(* IEC 61131-3 sources: Berechnungsplattform/PLC_CODESYS/Joystick, 2 files *)

(* ---- Gessmann_Joystick.st ---- *)
(* ============================================================================
   Gessmann Joystick / Thrust Lever CAN Interface
   Development Environment: CODESYS
   PLC Hardware: Intercontrol DIGSY Fusion S
   Description: Function block for reading Gessmann joystick and thrust lever
                signals via CAN bus
   ============================================================================ *)

TYPE Joystick_Axis :
STRUCT
    nRawValue       : INT;          (* Raw value from CAN message *)
    rScaledValue    : REAL;         (* Scaled value (-100.0 to +100.0 %) *)
    rDeadzone       : REAL := 5.0;  (* Deadzone in percent *)
    bInDeadzone     : BOOL;         (* Axis is in deadzone *)
    nMin            : INT := -32768;(* Minimum raw value *)
    nMax            : INT := 32767; (* Maximum raw value *)
    nCenter         : INT := 0;     (* Center/neutral raw value *)
END_STRUCT
END_TYPE

TYPE Gessmann_Joystick_Data :
STRUCT
    (* Axis data *)
    stAxisX         : Joystick_Axis;    (* X-Axis (left/right) *)
    stAxisY         : Joystick_Axis;    (* Y-Axis (forward/backward) *)
    stAxisZ         : Joystick_Axis;    (* Z-Axis / Twist (rotation) *)
    stThrustLever   : Joystick_Axis;    (* Thrust lever position *)

    (* Button states *)
    bButton1        : BOOL := FALSE;    (* Button 1 state *)
    bButton2        : BOOL := FALSE;    (* Button 2 state *)
    bButton3        : BOOL := FALSE;    (* Button 3 state *)
    bButton4        : BOOL := FALSE;    (* Button 4 state *)
    bButton5        : BOOL := FALSE;    (* Button 5 state *)
    bButton6        : BOOL := FALSE;    (* Button 6 state *)
    bButton7        : BOOL := FALSE;    (* Button 7 state *)
    bButton8        : BOOL := FALSE;    (* Button 8 state *)

    (* Status *)
    bOnline         : BOOL := FALSE;    (* Joystick communication active *)
    bError          : BOOL := FALSE;    (* Error flag *)
    dwErrorCode     : DWORD := 0;       (* Error code *)
END_STRUCT
END_TYPE

(* ============================================================================
   FUNCTION_BLOCK: FB_Gessmann_Joystick
   Description: Gessmann joystick/thrust lever handler via CAN
   ============================================================================ *)
FUNCTION_BLOCK FB_Gessmann_Joystick
VAR_INPUT
    bEnable             : BOOL := FALSE;        (* Enable joystick processing *)
    stCANMessage        : CAN_Message;          (* Incoming CAN message *)
    bNewCANMessage      : BOOL := FALSE;        (* New CAN message received *)
    dwJoystickCANID     : DWORD := 16#180;      (* Base CAN ID for joystick *)
    dwThrustLeverCANID  : DWORD := 16#181;      (* CAN ID for thrust lever *)
    dwButtonsCANID      : DWORD := 16#182;      (* CAN ID for buttons *)
    tTimeout            : TIME := T#500MS;      (* Communication timeout *)
    rDeadzoneX          : REAL := 5.0;          (* Deadzone for X-axis in % *)
    rDeadzoneY          : REAL := 5.0;          (* Deadzone for Y-axis in % *)
    rDeadzoneZ          : REAL := 5.0;          (* Deadzone for Z-axis in % *)
    rDeadzoneThrustLever: REAL := 2.0;          (* Deadzone for thrust lever in % *)
END_VAR

VAR_OUTPUT
    stJoystickData      : Gessmann_Joystick_Data;   (* Complete joystick data *)
    rAxisX              : REAL := 0.0;              (* X-Axis scaled output *)
    rAxisY              : REAL := 0.0;              (* Y-Axis scaled output *)
    rAxisZ              : REAL := 0.0;              (* Z-Axis scaled output *)
    rThrustLever        : REAL := 0.0;              (* Thrust lever scaled output *)
    bOnline             : BOOL := FALSE;            (* Communication status *)
    bError              : BOOL := FALSE;            (* Error flag *)
END_VAR

VAR
    tCommTimeout        : TON;                      (* Communication timeout timer *)
    bMessageReceived    : BOOL := FALSE;            (* Flag for received message *)
    dwLastMessageTime   : DWORD := 0;               (* Timestamp of last message *)
END_VAR

(* Main execution *)
IF NOT bEnable THEN
    (* Reset all outputs when disabled *)
    stJoystickData.bOnline := FALSE;
    bOnline := FALSE;
    rAxisX := 0.0;
    rAxisY := 0.0;
    rAxisZ := 0.0;
    rThrustLever := 0.0;
    RETURN;
END_IF

(* Set deadzone values *)
stJoystickData.stAxisX.rDeadzone := rDeadzoneX;
stJoystickData.stAxisY.rDeadzone := rDeadzoneY;
stJoystickData.stAxisZ.rDeadzone := rDeadzoneZ;
stJoystickData.stThrustLever.rDeadzone := rDeadzoneThrustLever;

(* Process incoming CAN messages *)
IF bNewCANMessage THEN
    bMessageReceived := TRUE;

    (* Process Joystick axes message *)
    IF stCANMessage.ID = dwJoystickCANID THEN
        (* Parse X-Axis from bytes 0-1 (high byte first)
           Using WORD intermediate to handle unsigned byte values correctly
           before converting to signed INT for the axis value *)
        stJoystickData.stAxisX.nRawValue := WORD_TO_INT(
            SHL(BYTE_TO_WORD(stCANMessage.Data[0]), 8)
            + BYTE_TO_WORD(stCANMessage.Data[1]));

        (* Parse Y-Axis from bytes 2-3 *)
        stJoystickData.stAxisY.nRawValue := WORD_TO_INT(
            SHL(BYTE_TO_WORD(stCANMessage.Data[2]), 8)
            + BYTE_TO_WORD(stCANMessage.Data[3]));

        (* Parse Z-Axis from bytes 4-5 *)
        stJoystickData.stAxisZ.nRawValue := WORD_TO_INT(
            SHL(BYTE_TO_WORD(stCANMessage.Data[4]), 8)
            + BYTE_TO_WORD(stCANMessage.Data[5]));

        (* Scale and apply deadzone to each axis *)
        ScaleAxis(stAxis := stJoystickData.stAxisX);
        ScaleAxis(stAxis := stJoystickData.stAxisY);
        ScaleAxis(stAxis := stJoystickData.stAxisZ);

        (* Update outputs *)
        rAxisX := stJoystickData.stAxisX.rScaledValue;
        rAxisY := stJoystickData.stAxisY.rScaledValue;
        rAxisZ := stJoystickData.stAxisZ.rScaledValue;

    (* Process Thrust Lever message *)
    ELSIF stCANMessage.ID = dwThrustLeverCANID THEN
        (* Parse Thrust Lever from bytes 0-1 *)
        stJoystickData.stThrustLever.nRawValue := WORD_TO_INT(
            SHL(BYTE_TO_WORD(stCANMessage.Data[0]), 8)
            + BYTE_TO_WORD(stCANMessage.Data[1]));

        (* Scale and apply deadzone *)
        ScaleAxis(stAxis := stJoystickData.stThrustLever);
        rThrustLever := stJoystickData.stThrustLever.rScaledValue;

    (* Process Buttons message *)
    ELSIF stCANMessage.ID = dwButtonsCANID THEN
        (* Parse button states from byte 0 *)
        stJoystickData.bButton1 := (stCANMessage.Data[0] AND 16#01) <> 0;
        stJoystickData.bButton2 := (stCANMessage.Data[0] AND 16#02) <> 0;
        stJoystickData.bButton3 := (stCANMessage.Data[0] AND 16#04) <> 0;
        stJoystickData.bButton4 := (stCANMessage.Data[0] AND 16#08) <> 0;
        stJoystickData.bButton5 := (stCANMessage.Data[0] AND 16#10) <> 0;
        stJoystickData.bButton6 := (stCANMessage.Data[0] AND 16#20) <> 0;
        stJoystickData.bButton7 := (stCANMessage.Data[0] AND 16#40) <> 0;
        stJoystickData.bButton8 := (stCANMessage.Data[0] AND 16#80) <> 0;
    END_IF

    (* Reset timeout timer on any valid message *)
    tCommTimeout(IN := FALSE);
END_IF

(* Communication timeout handling *)
tCommTimeout(IN := bEnable, PT := tTimeout);
IF tCommTimeout.Q THEN
    (* Timeout occurred - no message received within timeout period *)
    stJoystickData.bOnline := FALSE;
    stJoystickData.bError := TRUE;
    stJoystickData.dwErrorCode := 1; (* Timeout error *)
    bOnline := FALSE;
    bError := TRUE;

    (* Reset outputs to safe values *)
    rAxisX := 0.0;
    rAxisY := 0.0;
    rAxisZ := 0.0;
    rThrustLever := 0.0;
ELSE
    IF bMessageReceived THEN
        stJoystickData.bOnline := TRUE;
        stJoystickData.bError := FALSE;
        stJoystickData.dwErrorCode := 0;
        bOnline := TRUE;
        bError := FALSE;
    END_IF
END_IF

END_FUNCTION_BLOCK

(* ============================================================================
   ACTION: ScaleAxis
   Description: Scales raw joystick axis value to percentage and applies deadzone
   ============================================================================ *)
ACTION ScaleAxis
VAR_IN_OUT
    stAxis  : Joystick_Axis;
END_VAR

VAR
    rRawPercent : REAL;
    rRange      : REAL;
END_VAR

(* Calculate percentage from raw value *)
IF stAxis.nRawValue >= stAxis.nCenter THEN
    (* Positive direction *)
    rRange := INT_TO_REAL(stAxis.nMax - stAxis.nCenter);
    IF rRange > 0.0 THEN
        rRawPercent := INT_TO_REAL(stAxis.nRawValue - stAxis.nCenter) / rRange * 100.0;
    ELSE
        rRawPercent := 0.0;
    END_IF
ELSE
    (* Negative direction *)
    rRange := INT_TO_REAL(stAxis.nCenter - stAxis.nMin);
    IF rRange > 0.0 THEN
        rRawPercent := INT_TO_REAL(stAxis.nRawValue - stAxis.nCenter) / rRange * 100.0;
    ELSE
        rRawPercent := 0.0;
    END_IF
END_IF

(* Limit to valid range *)
IF rRawPercent > 100.0 THEN
    rRawPercent := 100.0;
ELSIF rRawPercent < -100.0 THEN
    rRawPercent := -100.0;
END_IF

(* Apply deadzone *)
IF ABS(rRawPercent) < stAxis.rDeadzone THEN
    stAxis.rScaledValue := 0.0;
    stAxis.bInDeadzone := TRUE;
ELSE
    (* Scale remaining range to full output range *)
    IF rRawPercent > 0.0 THEN
        stAxis.rScaledValue := (rRawPercent - stAxis.rDeadzone) / (100.0 - stAxis.rDeadzone) * 100.0;
    ELSE
        stAxis.rScaledValue := (rRawPercent + stAxis.rDeadzone) / (100.0 - stAxis.rDeadzone) * 100.0;
    END_IF
    stAxis.bInDeadzone := FALSE;
END_IF

END_ACTION

(* ---- Thrust_Lever_Control.st ---- *)
(* ============================================================================
   Thrust Lever Control Function Block
   Development Environment: CODESYS
   PLC Hardware: Intercontrol DIGSY Fusion S
   Description: Advanced thrust lever control with ramping, limits, and modes
   ============================================================================ *)

TYPE Thrust_Mode :
(
    THRUST_MODE_MANUAL := 0,        (* Direct joystick control *)
    THRUST_MODE_CRUISE := 1,        (* Cruise control / hold speed *)
    THRUST_MODE_RAMP := 2,          (* Ramped acceleration/deceleration *)
    THRUST_MODE_EMERGENCY := 3      (* Emergency stop *)
);
END_TYPE

TYPE Thrust_Status :
STRUCT
    eMode           : Thrust_Mode;      (* Current operating mode *)
    rCurrentThrust  : REAL;             (* Current thrust output (%) *)
    rTargetThrust   : REAL;             (* Target thrust (%) *)
    rRampRate       : REAL;             (* Current ramp rate (%/s) *)
    bLimitActive    : BOOL;             (* Limit is active *)
    bRamping        : BOOL;             (* Currently ramping *)
    bEmergency      : BOOL;             (* Emergency mode active *)
END_STRUCT
END_TYPE

(* ============================================================================
   FUNCTION_BLOCK: FB_Thrust_Lever_Control
   Description: Advanced thrust lever control with multiple operating modes
   ============================================================================ *)
FUNCTION_BLOCK FB_Thrust_Lever_Control
VAR_INPUT
    bEnable             : BOOL := FALSE;        (* Enable control *)
    rThrustLeverInput   : REAL := 0.0;          (* Raw thrust lever input (-100 to +100 %) *)
    eRequestedMode      : Thrust_Mode := THRUST_MODE_MANUAL;  (* Requested mode *)
    bEmergencyStop      : BOOL := FALSE;        (* Emergency stop trigger *)
    bCruiseSet          : BOOL := FALSE;        (* Set cruise control *)
    bCruiseResume       : BOOL := FALSE;        (* Resume cruise control *)
    bCruiseCancel       : BOOL := FALSE;        (* Cancel cruise control *)

    (* Configuration parameters *)
    rMaxThrust          : REAL := 100.0;        (* Maximum thrust limit (%) *)
    rMinThrust          : REAL := -100.0;       (* Minimum thrust limit (%) *)
    rRampUpRate         : REAL := 50.0;         (* Acceleration rate (%/s) *)
    rRampDownRate       : REAL := 75.0;         (* Deceleration rate (%/s) *)
    rEmergencyRampRate  : REAL := 200.0;        (* Emergency deceleration rate (%/s) *)
    rDeadband           : REAL := 2.0;          (* Input deadband (%) *)
    tCycleTime          : TIME := T#10MS;       (* PLC cycle time for rate calculations *)
END_VAR

VAR_OUTPUT
    rThrustOutput       : REAL := 0.0;          (* Final thrust output (-100 to +100 %) *)
    stStatus            : Thrust_Status;        (* Current status *)
    bActive             : BOOL := FALSE;        (* Control is active *)
    bAtTarget           : BOOL := FALSE;        (* Output equals target *)
END_VAR

VAR
    rInternalTarget     : REAL := 0.0;          (* Internal target thrust *)
    rInternalOutput     : REAL := 0.0;          (* Internal output value *)
    rCruiseSetpoint     : REAL := 0.0;          (* Stored cruise setpoint *)
    bCruiseActive       : BOOL := FALSE;        (* Cruise control is active *)
    rCycleTimeSeconds   : REAL := 0.01;         (* Cycle time in seconds *)
    rDelta              : REAL := 0.0;          (* Change per cycle *)
    bPrevCruiseSet      : BOOL := FALSE;        (* Previous cruise set state *)
END_VAR

(* Calculate cycle time in seconds *)
rCycleTimeSeconds := TIME_TO_REAL(tCycleTime) / 1000.0;

(* Main execution *)
IF NOT bEnable THEN
    rInternalOutput := 0.0;
    rInternalTarget := 0.0;
    rThrustOutput := 0.0;
    bActive := FALSE;
    stStatus.eMode := THRUST_MODE_MANUAL;
    stStatus.bEmergency := FALSE;
    bCruiseActive := FALSE;
    RETURN;
END_IF

bActive := TRUE;

(* Emergency stop handling - highest priority *)
IF bEmergencyStop THEN
    stStatus.eMode := THRUST_MODE_EMERGENCY;
    stStatus.bEmergency := TRUE;
    rInternalTarget := 0.0;
    bCruiseActive := FALSE;

    (* Fast ramp to zero *)
    IF rInternalOutput > 0.0 THEN
        rInternalOutput := rInternalOutput - (rEmergencyRampRate * rCycleTimeSeconds);
        IF rInternalOutput < 0.0 THEN
            rInternalOutput := 0.0;
        END_IF
    ELSIF rInternalOutput < 0.0 THEN
        rInternalOutput := rInternalOutput + (rEmergencyRampRate * rCycleTimeSeconds);
        IF rInternalOutput > 0.0 THEN
            rInternalOutput := 0.0;
        END_IF
    END_IF

ELSE
    stStatus.bEmergency := FALSE;

    (* Mode handling *)
    CASE eRequestedMode OF
        THRUST_MODE_MANUAL:
            stStatus.eMode := THRUST_MODE_MANUAL;
            bCruiseActive := FALSE;

            (* Apply deadband *)
            IF ABS(rThrustLeverInput) < rDeadband THEN
                rInternalTarget := 0.0;
            ELSE
                rInternalTarget := rThrustLeverInput;
            END_IF

            (* Apply limits *)
            IF rInternalTarget > rMaxThrust THEN
                rInternalTarget := rMaxThrust;
                stStatus.bLimitActive := TRUE;
            ELSIF rInternalTarget < rMinThrust THEN
                rInternalTarget := rMinThrust;
                stStatus.bLimitActive := TRUE;
            ELSE
                stStatus.bLimitActive := FALSE;
            END_IF

            (* Direct output in manual mode *)
            rInternalOutput := rInternalTarget;

        THRUST_MODE_CRUISE:
            stStatus.eMode := THRUST_MODE_CRUISE;

            (* Cruise set button rising edge *)
            IF bCruiseSet AND NOT bPrevCruiseSet THEN
                rCruiseSetpoint := rInternalOutput;
                bCruiseActive := TRUE;
            END_IF
            bPrevCruiseSet := bCruiseSet;

            (* Resume cruise *)
            IF bCruiseResume AND rCruiseSetpoint <> 0.0 THEN
                bCruiseActive := TRUE;
            END_IF

            (* Cancel cruise *)
            IF bCruiseCancel THEN
                bCruiseActive := FALSE;
            END_IF

            (* Cruise operation *)
            IF bCruiseActive THEN
                rInternalTarget := rCruiseSetpoint;
            ELSE
                (* Fall back to manual input if cruise not active *)
                IF ABS(rThrustLeverInput) < rDeadband THEN
                    rInternalTarget := 0.0;
                ELSE
                    rInternalTarget := rThrustLeverInput;
                END_IF
            END_IF

            (* Ramp to target *)
            RampToTarget();

        THRUST_MODE_RAMP:
            stStatus.eMode := THRUST_MODE_RAMP;
            bCruiseActive := FALSE;

            (* Apply deadband *)
            IF ABS(rThrustLeverInput) < rDeadband THEN
                rInternalTarget := 0.0;
            ELSE
                rInternalTarget := rThrustLeverInput;
            END_IF

            (* Apply limits *)
            IF rInternalTarget > rMaxThrust THEN
                rInternalTarget := rMaxThrust;
                stStatus.bLimitActive := TRUE;
            ELSIF rInternalTarget < rMinThrust THEN
                rInternalTarget := rMinThrust;
                stStatus.bLimitActive := TRUE;
            ELSE
                stStatus.bLimitActive := FALSE;
            END_IF

            (* Ramp to target *)
            RampToTarget();

        ELSE
            (* Unknown mode - default to manual *)
            stStatus.eMode := THRUST_MODE_MANUAL;
            rInternalOutput := rThrustLeverInput;
    END_CASE
END_IF

(* Update status *)
stStatus.rCurrentThrust := rInternalOutput;
stStatus.rTargetThrust := rInternalTarget;
bAtTarget := ABS(rInternalOutput - rInternalTarget) < 0.1;

(* Set output *)
rThrustOutput := rInternalOutput;

END_FUNCTION_BLOCK

(* ============================================================================
   ACTION: RampToTarget
   Description: Ramps output towards target with configurable rates
   ============================================================================ *)
ACTION RampToTarget

(* Calculate required change *)
rDelta := rInternalTarget - rInternalOutput;

IF ABS(rDelta) < 0.1 THEN
    (* Close enough - snap to target *)
    rInternalOutput := rInternalTarget;
    stStatus.bRamping := FALSE;
    stStatus.rRampRate := 0.0;
ELSE
    stStatus.bRamping := TRUE;

    IF rDelta > 0.0 THEN
        (* Ramping up (accelerating) *)
        stStatus.rRampRate := rRampUpRate;
        rInternalOutput := rInternalOutput + (rRampUpRate * rCycleTimeSeconds);
        IF rInternalOutput > rInternalTarget THEN
            rInternalOutput := rInternalTarget;
        END_IF
    ELSE
        (* Ramping down (decelerating) *)
        stStatus.rRampRate := rRampDownRate;
        rInternalOutput := rInternalOutput - (rRampDownRate * rCycleTimeSeconds);
        IF rInternalOutput < rInternalTarget THEN
            rInternalOutput := rInternalTarget;
        END_IF
    END_IF
END_IF

END_ACTION
